(* Logix 5000 project; controller SX_V040001_C001 vendor 1 type 14 code 77 rev 16.23; software revision 16.04; part 4 of 35 *)
(* tags used below, declared in another part *)
   ALARM_BITS : INT[10];
   ALL_KINDS : INT[90];
   Basic : INT;
   DRIVE : INT[32];
   EMPTYING : INT[18];
   G_DInput : DINT[3];
   G_DOutput : DINT[3];
   louvre : INT[11];
   m_alarm_exist : BOOL;
   m_notstop : BOOL;
   METERING : INT[44];
   PARAMETER : INT[501];
   T_AIR_EXH_FAN : TIMER;
   T_AIR_IN_FAN : TIMER;
   T_AIR_IN_HEATING : TIMER;
   T_CHOCO_PUMP : TIMER;
   T_COVER_DOM : TIMER;
   T_ELEKTR_HEAT : TIMER;
   T_INTERN_CIRCLE : TIMER;
   T_LOUVRE : TIMER;
   T_MET5_END : TIMER;
   T_OUTLETT_VALVE : TIMER;
   T_SAMPLER_OPEN : TIMER;
   T_WATER_NIVEAU : TIMER;
   T_WATERPUMP : TIMER;
   TEMP : INT[14];
   Z15 : COUNTER;
   Z16 : COUNTER;
   Z17 : COUNTER;
   Z18 : COUNTER;
   Z29 : COUNTER;
   Z32 : COUNTER;
(* MainProgram, continued *)

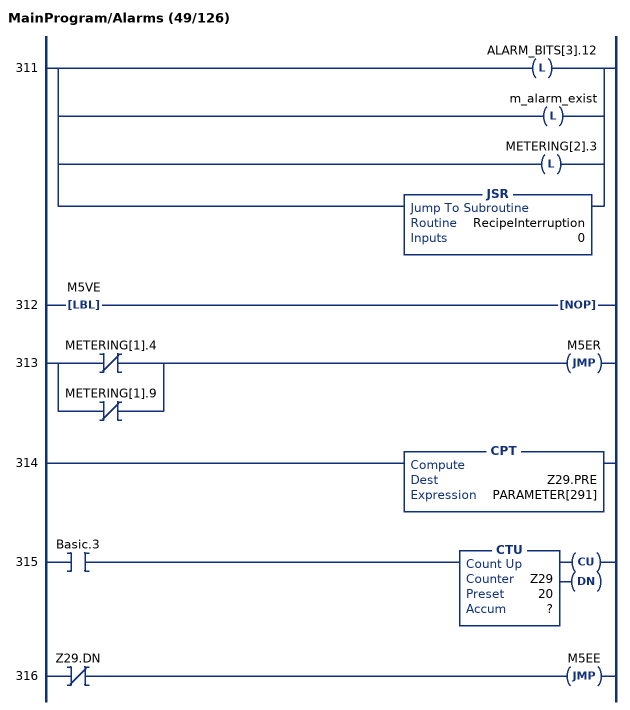
   [picture p70: MainProgram/Alarms rungs 311-316]
   311: [OTL(ALARM_BITS[3].12) ,OTL(m_alarm_exist) ,OTL(METERING[2].3) ,JSR(RecipeInterruption,0) ];
   312: LBL(M5VE)NOP();
   313: [XIO(METERING[1].4) ,XIO(METERING[1].9) ]JMP(M5ER);
   314: CPT(Z29.PRE,PARAMETER[291]);
   315: XIC(Basic.3)CTU(Z29,?,?);
   316: XIO(Z29.DN)JMP(M5EE);
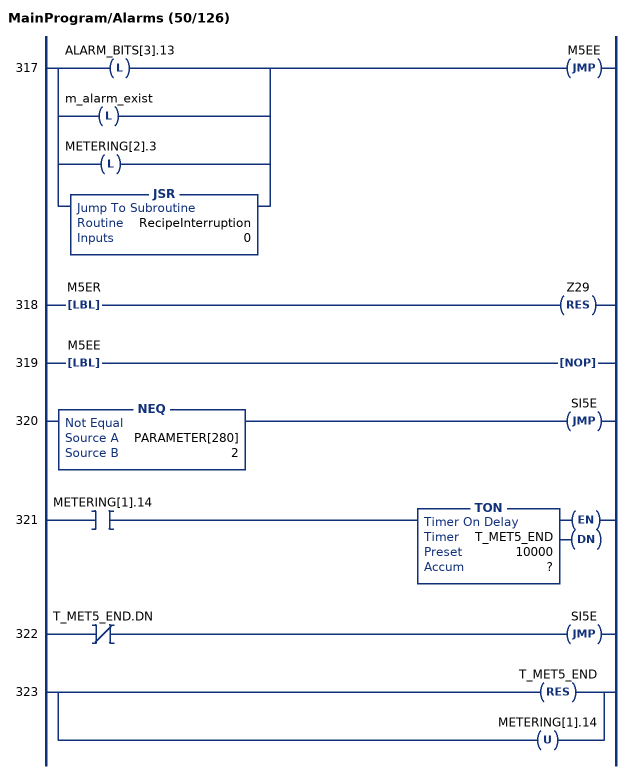
   317: [OTL(ALARM_BITS[3].13) ,OTL(m_alarm_exist) ,OTL(METERING[2].3) ,JSR(RecipeInterruption,0) ]JMP(M5EE);
   318: LBL(M5ER)RES(Z29);
   319: LBL(M5EE)NOP();
   320: NEQ(PARAMETER[280],2)JMP(SI5E);
   321: XIC(METERING[1].14)TON(T_MET5_END,?,?);
   322: XIO(T_MET5_END.DN)JMP(SI5E);
   323: [RES(T_MET5_END) ,OTU(METERING[1].14) ];
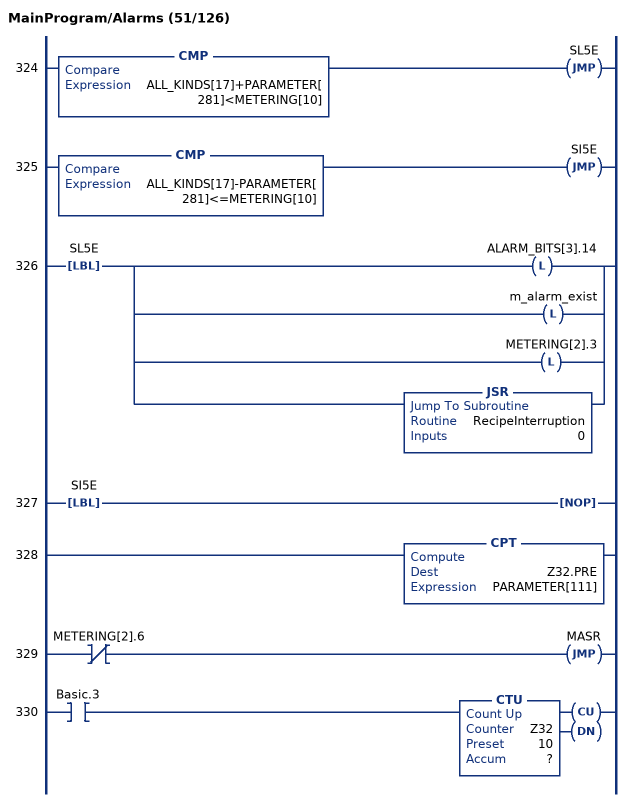
   324: CMP(ALL_KINDS[17]+PARAMETER[281]<METERING[10])JMP(SL5E);
   325: CMP(ALL_KINDS[17]-PARAMETER[281]<=METERING[10])JMP(SI5E);
   326: LBL(SL5E)[OTL(ALARM_BITS[3].14) ,OTL(m_alarm_exist) ,OTL(METERING[2].3) ,JSR(RecipeInterruption,0) ];
   327: LBL(SI5E)NOP();
   328: CPT(Z32.PRE,PARAMETER[111]);
   329: XIO(METERING[2].6)JMP(MASR);
   330: XIC(Basic.3)CTU(Z32,?,?);
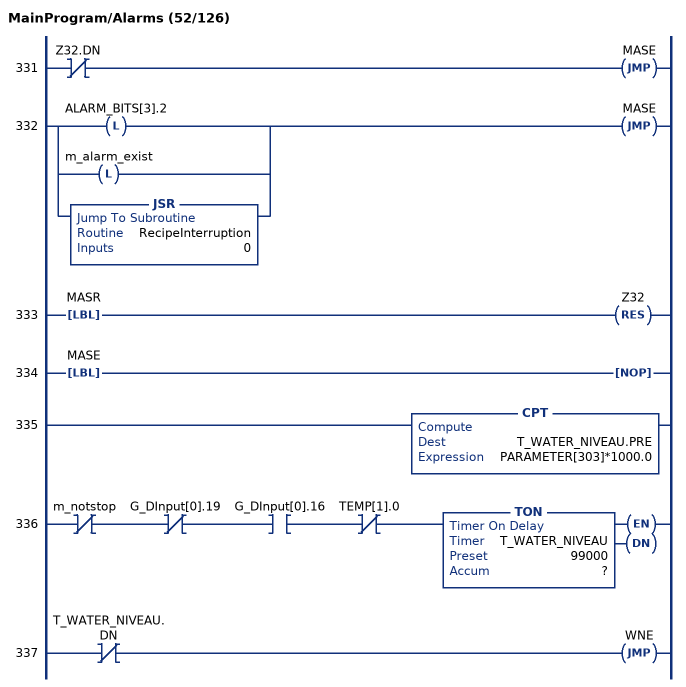
   331: XIO(Z32.DN)JMP(MASE);
   332: [OTL(ALARM_BITS[3].2) ,OTL(m_alarm_exist) ,JSR(RecipeInterruption,0) ]JMP(MASE);
   333: LBL(MASR)RES(Z32);
   334: LBL(MASE)NOP();
   335: CPT(T_WATER_NIVEAU.PRE,PARAMETER[303]*1000.0);
   336: XIO(m_notstop)XIO(G_DInput[0].19)XIC(G_DInput[0].16)XIO(TEMP[1].0)TON(T_WATER_NIVEAU,?,?);
   337: XIO(T_WATER_NIVEAU.DN)JMP(WNE);
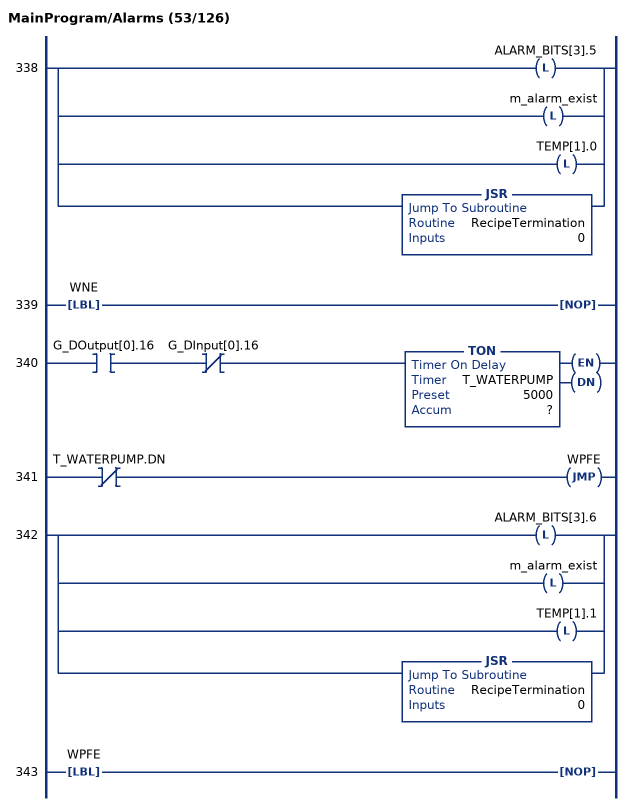
   338: [OTL(ALARM_BITS[3].5) ,OTL(m_alarm_exist) ,OTL(TEMP[1].0) ,JSR(RecipeTermination,0) ];
   339: LBL(WNE)NOP();
   340: XIC(G_DOutput[0].16)XIO(G_DInput[0].16)TON(T_WATERPUMP,?,?);
   341: XIO(T_WATERPUMP.DN)JMP(WPFE);
   342: [OTL(ALARM_BITS[3].6) ,OTL(m_alarm_exist) ,OTL(TEMP[1].1) ,JSR(RecipeTermination,0) ];
   343: LBL(WPFE)NOP();
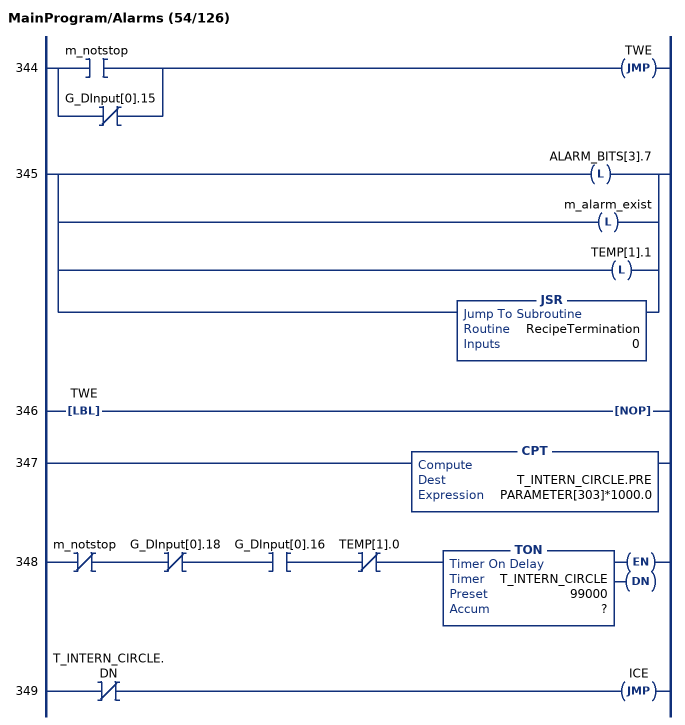
   344: [XIC(m_notstop) ,XIO(G_DInput[0].15) ]JMP(TWE);
   345: [OTL(ALARM_BITS[3].7) ,OTL(m_alarm_exist) ,OTL(TEMP[1].1) ,JSR(RecipeTermination,0) ];
   346: LBL(TWE)NOP();
   347: CPT(T_INTERN_CIRCLE.PRE,PARAMETER[303]*1000.0);
   348: XIO(m_notstop)XIO(G_DInput[0].18)XIC(G_DInput[0].16)XIO(TEMP[1].0)TON(T_INTERN_CIRCLE,?,?);
   349: XIO(T_INTERN_CIRCLE.DN)JMP(ICE);
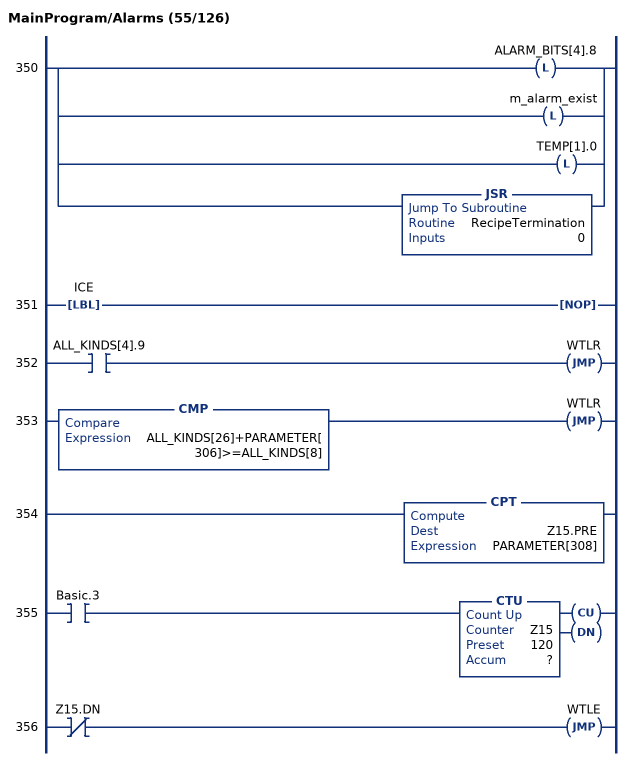
   350: [OTL(ALARM_BITS[4].8) ,OTL(m_alarm_exist) ,OTL(TEMP[1].0) ,JSR(RecipeTermination,0) ];
   351: LBL(ICE)NOP();
   352: XIC(ALL_KINDS[4].9)JMP(WTLR);
   353: CMP(ALL_KINDS[26]+PARAMETER[306]>=ALL_KINDS[8])JMP(WTLR);
   354: CPT(Z15.PRE,PARAMETER[308]);
   355: XIC(Basic.3)CTU(Z15,?,?);
   356: XIO(Z15.DN)JMP(WTLE);
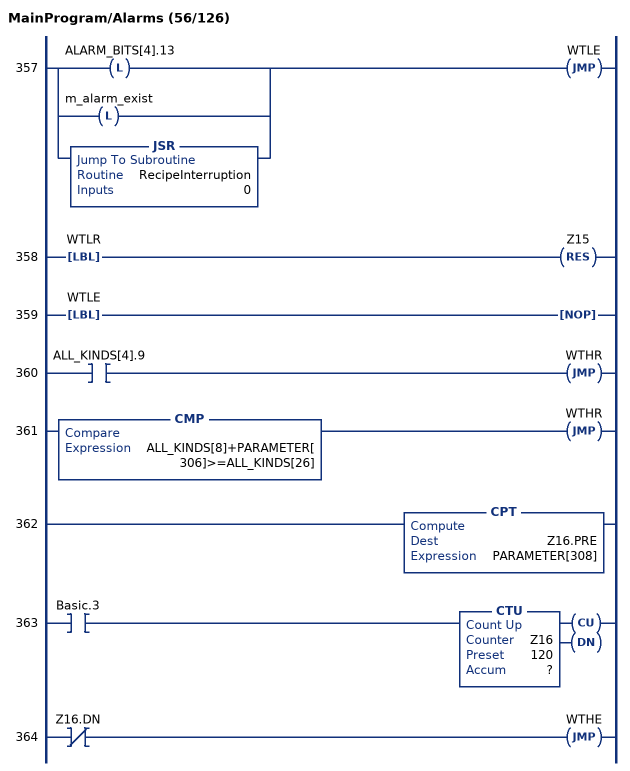
   357: [OTL(ALARM_BITS[4].13) ,OTL(m_alarm_exist) ,JSR(RecipeInterruption,0) ]JMP(WTLE);
   358: LBL(WTLR)RES(Z15);
   359: LBL(WTLE)NOP();
   360: XIC(ALL_KINDS[4].9)JMP(WTHR);
   361: CMP(ALL_KINDS[8]+PARAMETER[306]>=ALL_KINDS[26])JMP(WTHR);
   362: CPT(Z16.PRE,PARAMETER[308]);
   363: XIC(Basic.3)CTU(Z16,?,?);
   364: XIO(Z16.DN)JMP(WTHE);
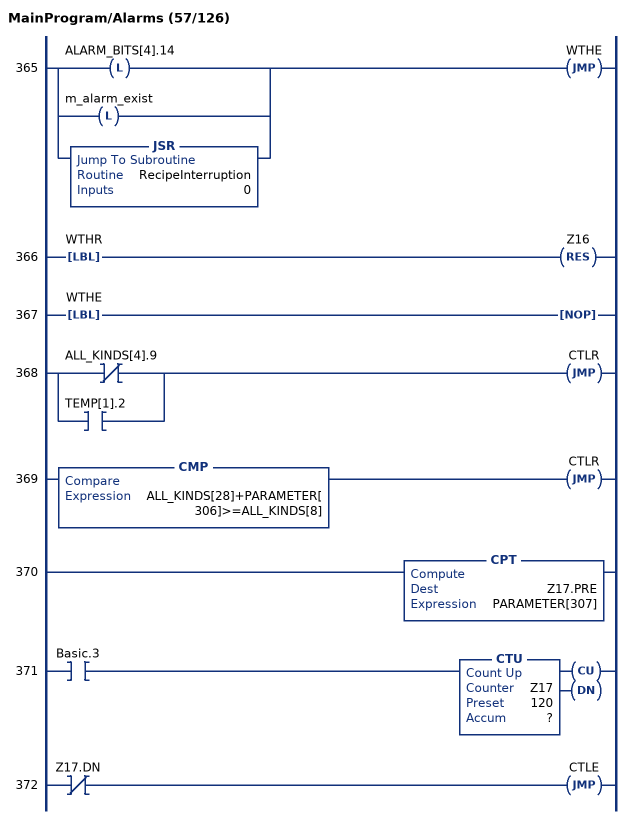
   365: [OTL(ALARM_BITS[4].14) ,OTL(m_alarm_exist) ,JSR(RecipeInterruption,0) ]JMP(WTHE);
   366: LBL(WTHR)RES(Z16);
   367: LBL(WTHE)NOP();
   368: [XIO(ALL_KINDS[4].9) ,XIC(TEMP[1].2) ]JMP(CTLR);
   369: CMP(ALL_KINDS[28]+PARAMETER[306]>=ALL_KINDS[8])JMP(CTLR);
   370: CPT(Z17.PRE,PARAMETER[307]);
   371: XIC(Basic.3)CTU(Z17,?,?);
   372: XIO(Z17.DN)JMP(CTLE);
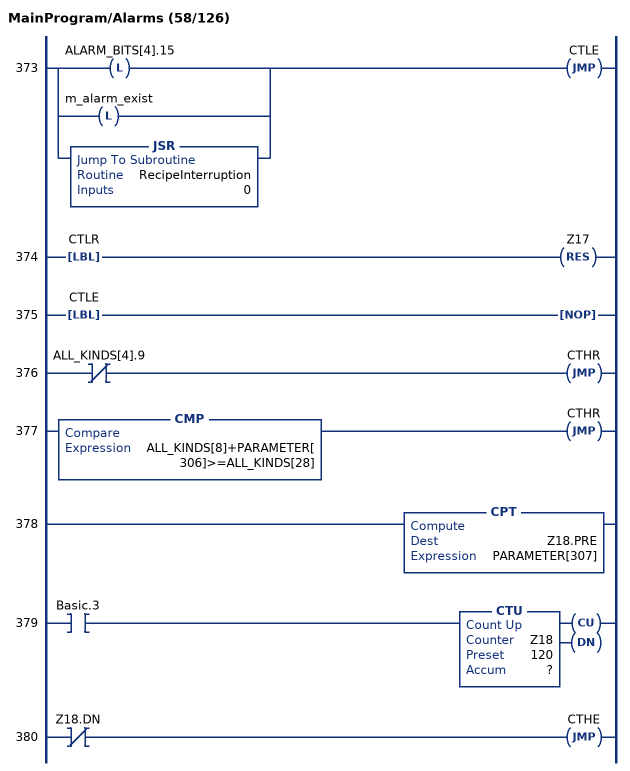
   373: [OTL(ALARM_BITS[4].15) ,OTL(m_alarm_exist) ,JSR(RecipeInterruption,0) ]JMP(CTLE);
   374: LBL(CTLR)RES(Z17);
   375: LBL(CTLE)NOP();
   376: XIO(ALL_KINDS[4].9)JMP(CTHR);
   377: CMP(ALL_KINDS[8]+PARAMETER[306]>=ALL_KINDS[28])JMP(CTHR);
   378: CPT(Z18.PRE,PARAMETER[307]);
   379: XIC(Basic.3)CTU(Z18,?,?);
   380: XIO(Z18.DN)JMP(CTHE);
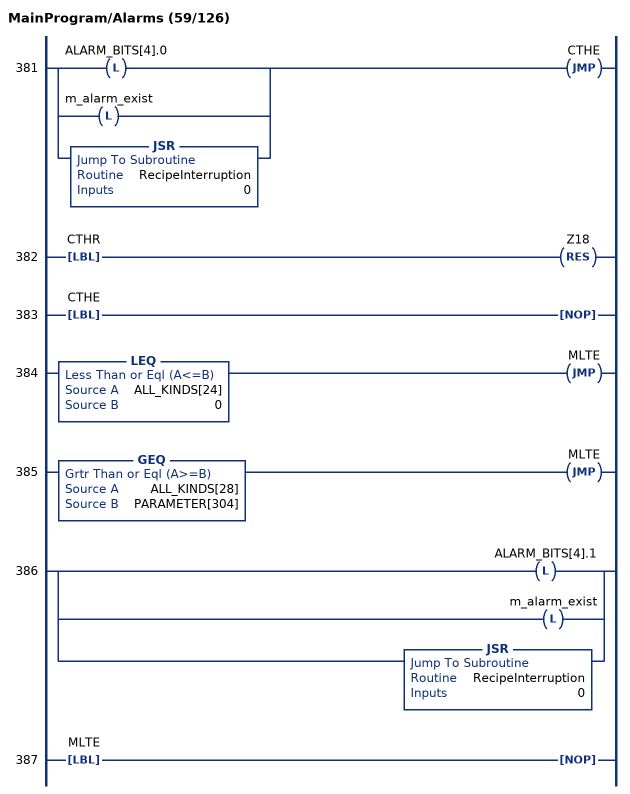
   381: [OTL(ALARM_BITS[4].0) ,OTL(m_alarm_exist) ,JSR(RecipeInterruption,0) ]JMP(CTHE);
   382: LBL(CTHR)RES(Z18);
   383: LBL(CTHE)NOP();
   384: LEQ(ALL_KINDS[24],0)JMP(MLTE);
   385: GEQ(ALL_KINDS[28],PARAMETER[304])JMP(MLTE);
   386: [OTL(ALARM_BITS[4].1) ,OTL(m_alarm_exist) ,JSR(RecipeInterruption,0) ];
   387: LBL(MLTE)NOP();
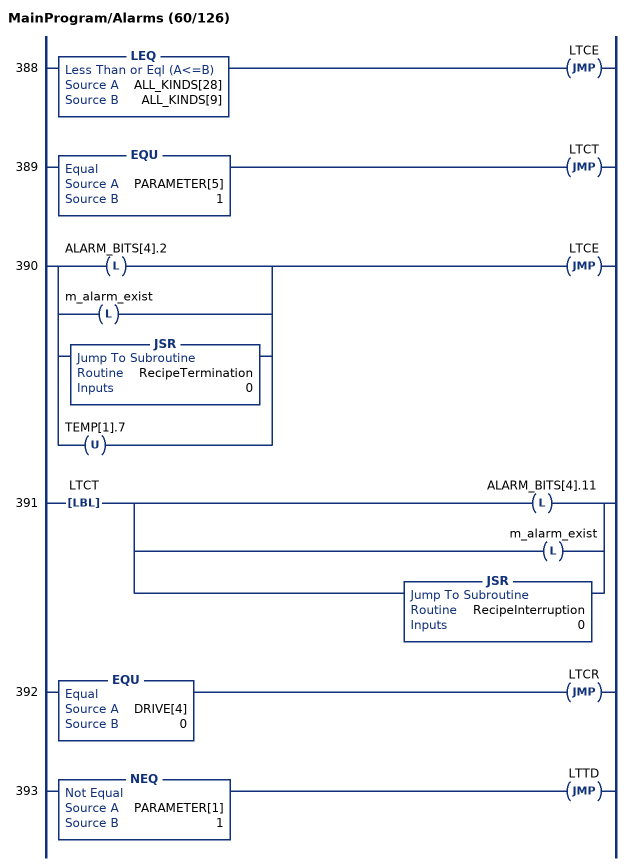
   388: LEQ(ALL_KINDS[28],ALL_KINDS[9])JMP(LTCE);
   389: EQU(PARAMETER[5],1)JMP(LTCT);
   390: [OTL(ALARM_BITS[4].2) ,OTL(m_alarm_exist) ,JSR(RecipeTermination,0) ,OTU(TEMP[1].7) ]JMP(LTCE);
   391: LBL(LTCT)[OTL(ALARM_BITS[4].11) ,OTL(m_alarm_exist) ,JSR(RecipeInterruption,0) ];
   392: EQU(DRIVE[4],0)JMP(LTCR);
   393: NEQ(PARAMETER[1],1)JMP(LTTD);
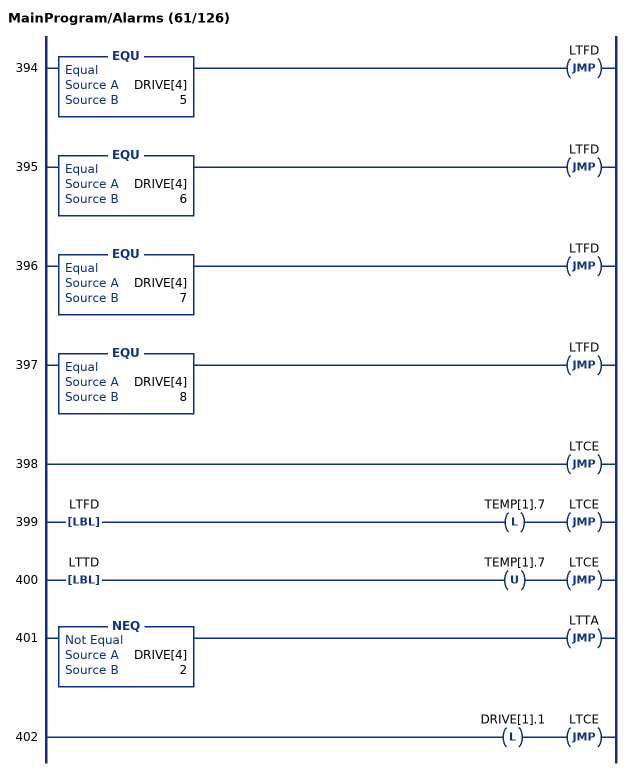
   394: EQU(DRIVE[4],5)JMP(LTFD);
   395: EQU(DRIVE[4],6)JMP(LTFD);
   396: EQU(DRIVE[4],7)JMP(LTFD);
   397: EQU(DRIVE[4],8)JMP(LTFD);
   398: JMP(LTCE);
   399: LBL(LTFD)OTL(TEMP[1].7)JMP(LTCE);
   400: LBL(LTTD)OTU(TEMP[1].7)JMP(LTCE);
   401: NEQ(DRIVE[4],2)JMP(LTTA);
   402: OTL(DRIVE[1].1)JMP(LTCE);
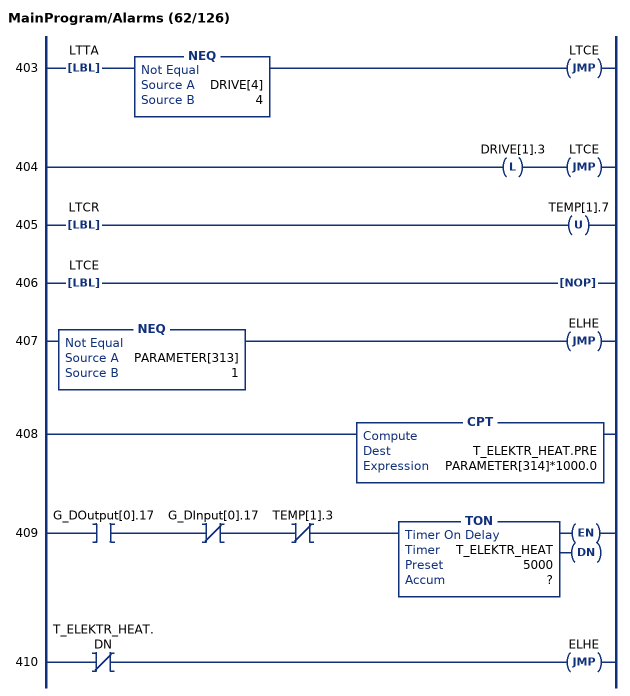
   403: LBL(LTTA)NEQ(DRIVE[4],4)JMP(LTCE);
   404: OTL(DRIVE[1].3)JMP(LTCE);
   405: LBL(LTCR)OTU(TEMP[1].7);
   406: LBL(LTCE)NOP();
   407: NEQ(PARAMETER[313],1)JMP(ELHE);
   408: CPT(T_ELEKTR_HEAT.PRE,PARAMETER[314]*1000.0);
   409: XIC(G_DOutput[0].17)XIO(G_DInput[0].17)XIO(TEMP[1].3)TON(T_ELEKTR_HEAT,?,?);
   410: XIO(T_ELEKTR_HEAT.DN)JMP(ELHE);
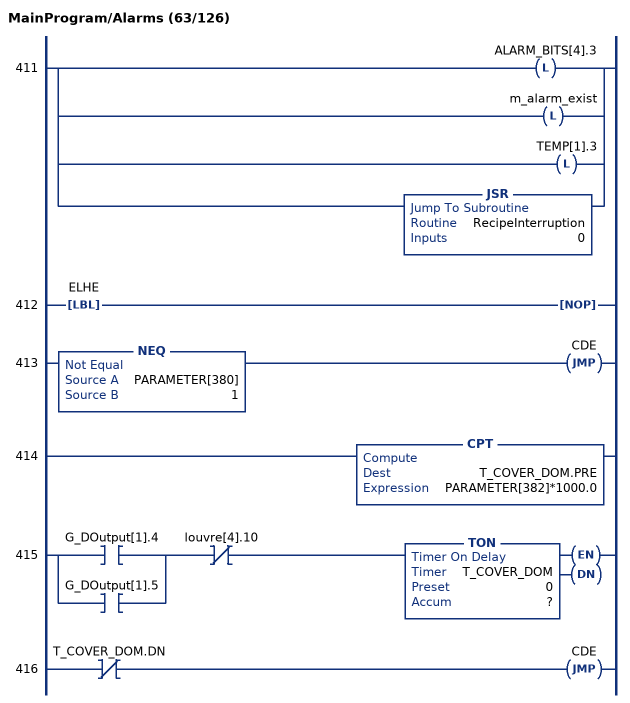
   411: [OTL(ALARM_BITS[4].3) ,OTL(m_alarm_exist) ,OTL(TEMP[1].3) ,JSR(RecipeInterruption,0) ];
   412: LBL(ELHE)NOP();
   413: NEQ(PARAMETER[380],1)JMP(CDE);
   414: CPT(T_COVER_DOM.PRE,PARAMETER[382]*1000.0);
   415: [XIC(G_DOutput[1].4) ,XIC(G_DOutput[1].5) ]XIO(louvre[4].10)TON(T_COVER_DOM,?,?);
   416: XIO(T_COVER_DOM.DN)JMP(CDE);
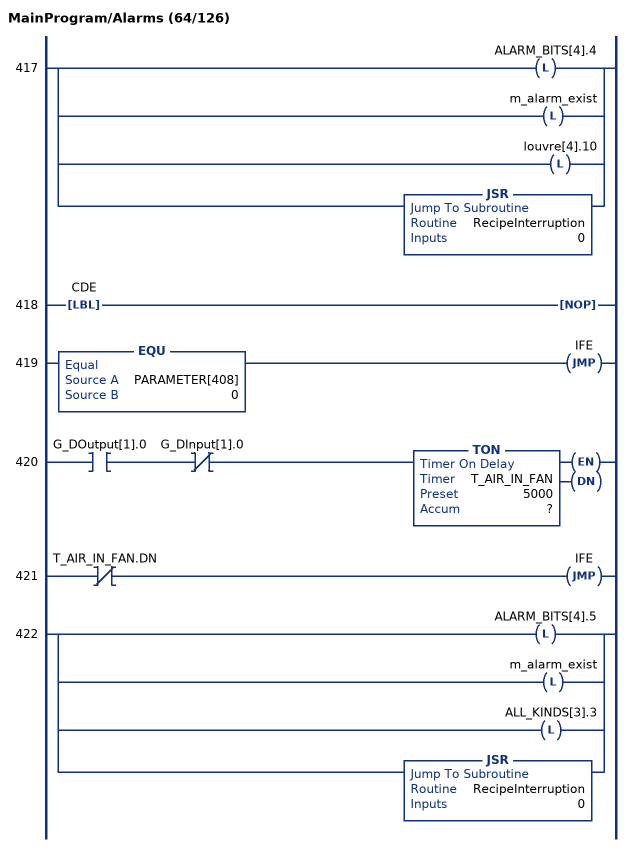
   417: [OTL(ALARM_BITS[4].4) ,OTL(m_alarm_exist) ,OTL(louvre[4].10) ,JSR(RecipeInterruption,0) ];
   418: LBL(CDE)NOP();
   419: EQU(PARAMETER[408],0)JMP(IFE);
   420: XIC(G_DOutput[1].0)XIO(G_DInput[1].0)TON(T_AIR_IN_FAN,?,?);
   421: XIO(T_AIR_IN_FAN.DN)JMP(IFE);
   422: [OTL(ALARM_BITS[4].5) ,OTL(m_alarm_exist) ,OTL(ALL_KINDS[3].3) ,JSR(RecipeInterruption,0) ];
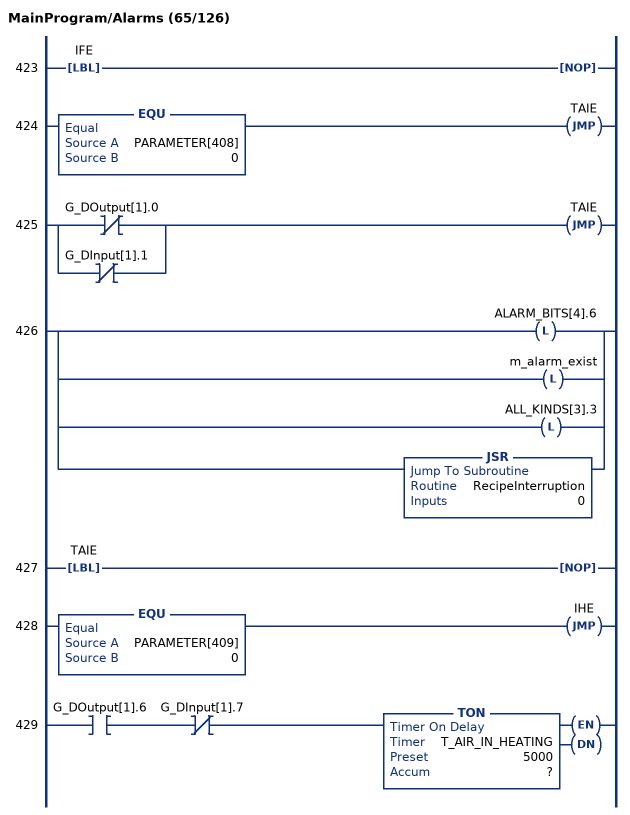
   423: LBL(IFE)NOP();
   424: EQU(PARAMETER[408],0)JMP(TAIE);
   425: [XIO(G_DOutput[1].0) ,XIO(G_DInput[1].1) ]JMP(TAIE);
   426: [OTL(ALARM_BITS[4].6) ,OTL(m_alarm_exist) ,OTL(ALL_KINDS[3].3) ,JSR(RecipeInterruption,0) ];
   427: LBL(TAIE)NOP();
   428: EQU(PARAMETER[409],0)JMP(IHE);
   429: XIC(G_DOutput[1].6)XIO(G_DInput[1].7)TON(T_AIR_IN_HEATING,?,?);
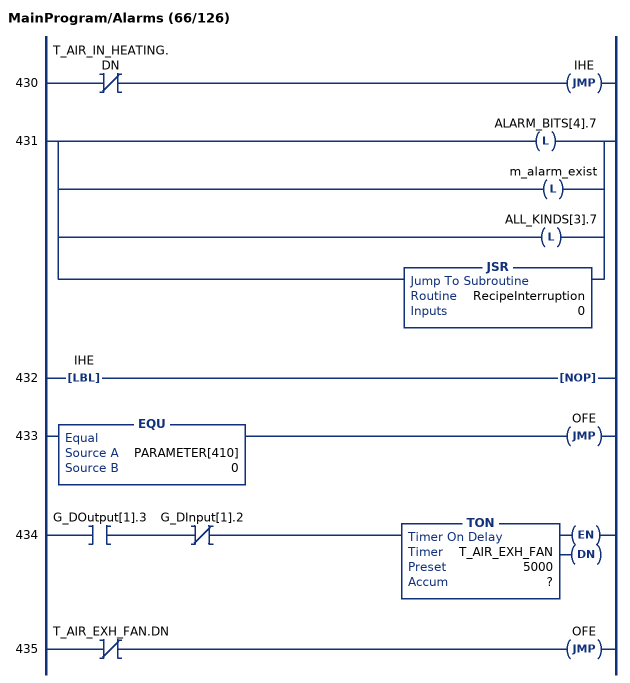
   430: XIO(T_AIR_IN_HEATING.DN)JMP(IHE);
   431: [OTL(ALARM_BITS[4].7) ,OTL(m_alarm_exist) ,OTL(ALL_KINDS[3].7) ,JSR(RecipeInterruption,0) ];
   432: LBL(IHE)NOP();
   433: EQU(PARAMETER[410],0)JMP(OFE);
   434: XIC(G_DOutput[1].3)XIO(G_DInput[1].2)TON(T_AIR_EXH_FAN,?,?);
   435: XIO(T_AIR_EXH_FAN.DN)JMP(OFE);
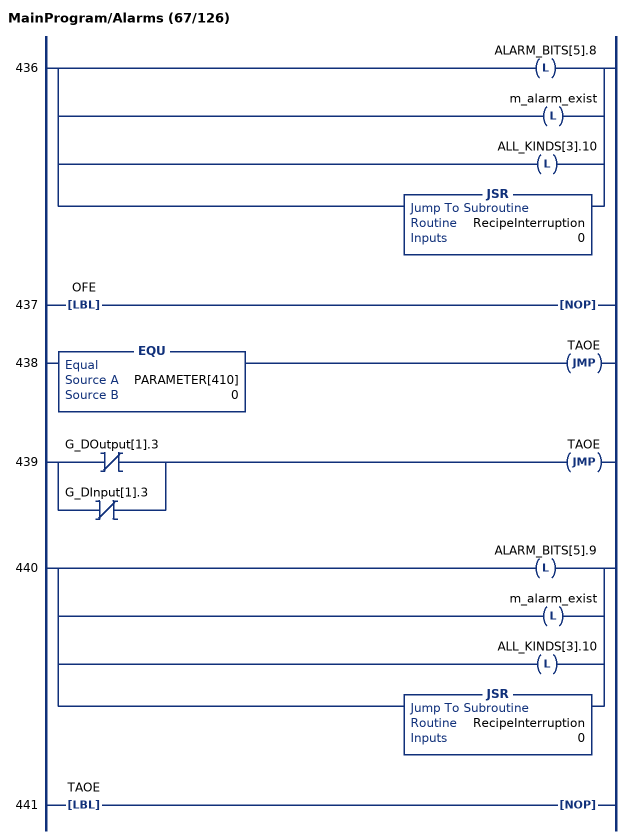
   436: [OTL(ALARM_BITS[5].8) ,OTL(m_alarm_exist) ,OTL(ALL_KINDS[3].10) ,JSR(RecipeInterruption,0) ];
   437: LBL(OFE)NOP();
   438: EQU(PARAMETER[410],0)JMP(TAOE);
   439: [XIO(G_DOutput[1].3) ,XIO(G_DInput[1].3) ]JMP(TAOE);
   440: [OTL(ALARM_BITS[5].9) ,OTL(m_alarm_exist) ,OTL(ALL_KINDS[3].10) ,JSR(RecipeInterruption,0) ];
   441: LBL(TAOE)NOP();
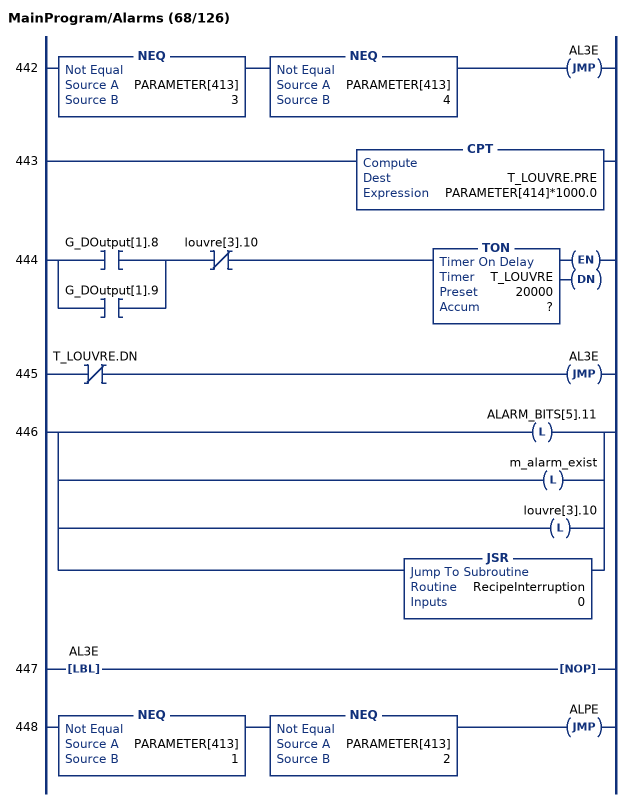
   442: NEQ(PARAMETER[413],3)NEQ(PARAMETER[413],4)JMP(AL3E);
   443: CPT(T_LOUVRE.PRE,PARAMETER[414]*1000.0);
   444: [XIC(G_DOutput[1].8) ,XIC(G_DOutput[1].9) ]XIO(louvre[3].10)TON(T_LOUVRE,?,?);
   445: XIO(T_LOUVRE.DN)JMP(AL3E);
   446: [OTL(ALARM_BITS[5].11) ,OTL(m_alarm_exist) ,OTL(louvre[3].10) ,JSR(RecipeInterruption,0) ];
   447: LBL(AL3E)NOP();
   448: NEQ(PARAMETER[413],1)NEQ(PARAMETER[413],2)JMP(ALPE);
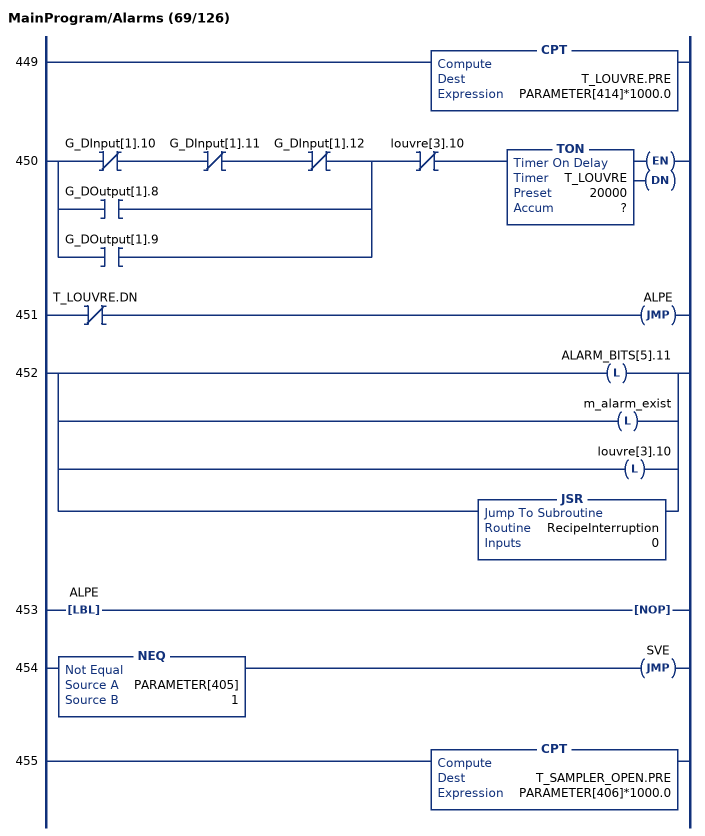
   449: CPT(T_LOUVRE.PRE,PARAMETER[414]*1000.0);
   450: [XIO(G_DInput[1].10) XIO(G_DInput[1].11) XIO(G_DInput[1].12) ,XIC(G_DOutput[1].8) ,XIC(G_DOutput[1].9) ]XIO(louvre[3].10)TON(T_LOUVRE,?,?);
   451: XIO(T_LOUVRE.DN)JMP(ALPE);
   452: [OTL(ALARM_BITS[5].11) ,OTL(m_alarm_exist) ,OTL(louvre[3].10) ,JSR(RecipeInterruption,0) ];
   453: LBL(ALPE)NOP();
   454: NEQ(PARAMETER[405],1)JMP(SVE);
   455: CPT(T_SAMPLER_OPEN.PRE,PARAMETER[406]*1000.0);
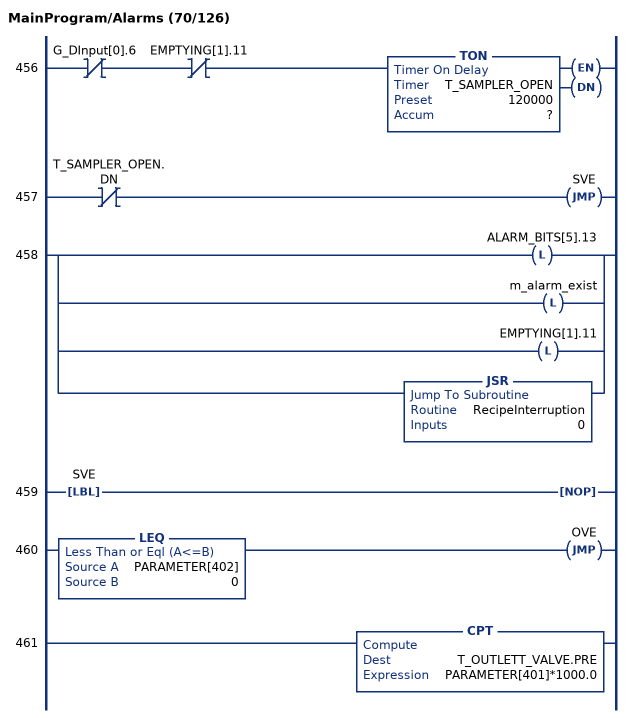
   456: XIO(G_DInput[0].6)XIO(EMPTYING[1].11)TON(T_SAMPLER_OPEN,?,?);
   457: XIO(T_SAMPLER_OPEN.DN)JMP(SVE);
   458: [OTL(ALARM_BITS[5].13) ,OTL(m_alarm_exist) ,OTL(EMPTYING[1].11) ,JSR(RecipeInterruption,0) ];
   459: LBL(SVE)NOP();
   460: LEQ(PARAMETER[402],0)JMP(OVE);
   461: CPT(T_OUTLETT_VALVE.PRE,PARAMETER[401]*1000.0);
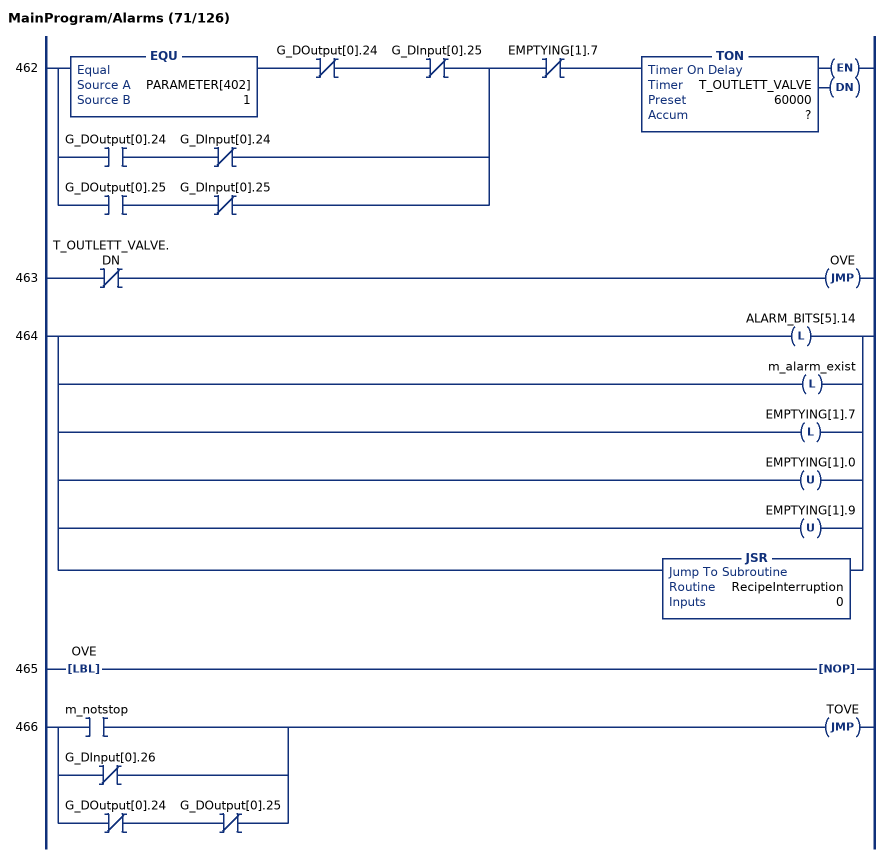
   462: [EQU(PARAMETER[402],1) XIO(G_DOutput[0].24) XIO(G_DInput[0].25) ,XIC(G_DOutput[0].24) XIO(G_DInput[0].24) ,XIC(G_DOutput[0].25) XIO(G_DInput[0].25) ]XIO(EMPTYING[1].7)TON(T_OUTLETT_VALVE,?,?);
   463: XIO(T_OUTLETT_VALVE.DN)JMP(OVE);
   464: [OTL(ALARM_BITS[5].14) ,OTL(m_alarm_exist) ,OTL(EMPTYING[1].7) ,OTU(EMPTYING[1].0) ,OTU(EMPTYING[1].9) ,JSR(RecipeInterruption,0) ];
   465: LBL(OVE)NOP();
   466: [XIC(m_notstop) ,XIO(G_DInput[0].26) ,XIO(G_DOutput[0].24) XIO(G_DOutput[0].25) ]JMP(TOVE);
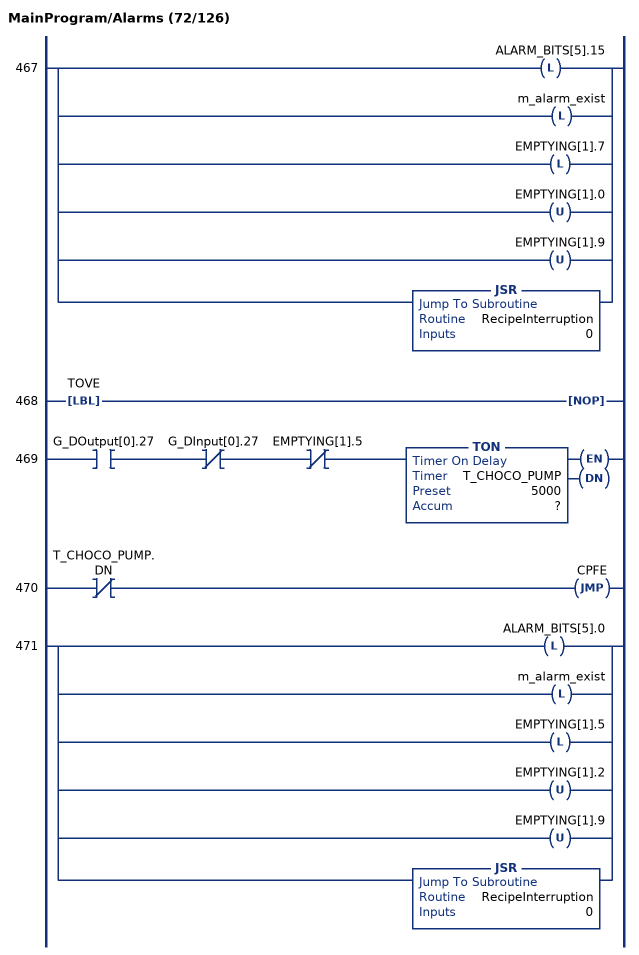
   467: [OTL(ALARM_BITS[5].15) ,OTL(m_alarm_exist) ,OTL(EMPTYING[1].7) ,OTU(EMPTYING[1].0) ,OTU(EMPTYING[1].9) ,JSR(RecipeInterruption,0) ];
   468: LBL(TOVE)NOP();
   469: XIC(G_DOutput[0].27)XIO(G_DInput[0].27)XIO(EMPTYING[1].5)TON(T_CHOCO_PUMP,?,?);
   470: XIO(T_CHOCO_PUMP.DN)JMP(CPFE);
   471: [OTL(ALARM_BITS[5].0) ,OTL(m_alarm_exist) ,OTL(EMPTYING[1].5) ,OTU(EMPTYING[1].2) ,OTU(EMPTYING[1].9) ,JSR(RecipeInterruption,0) ];
